SYSTEM TestFirstAgentFB (* System Configuration *)
  (* Standard: 61499-1 *)
  (* Version 0.3, 2003-12-05, JHC, Rockwell Automation, Renamed from NEWSYSTEM. *)
  (* Version 0.2, 2002-11-05, JHC, Rockwell Automation, Fixed missing (empty) FBD in Application. *)
  (* Version 0.1, 2002-01-17, JHC, Rockwell Automation, Minor cleanup *)
  (* Version 0.0, 2000-05-27, JHC, Rockwell Automation *)
  APPLICATION APP1
  END_APPLICATION
  DEVICE MyPLC : FRAME_DEVICE(BOUNDS := [1100,100,500,500], GRID := [1,1])
    RESOURCE MyProcessor : PANEL_RESOURCE(ROWS := 4, COLS := 4)
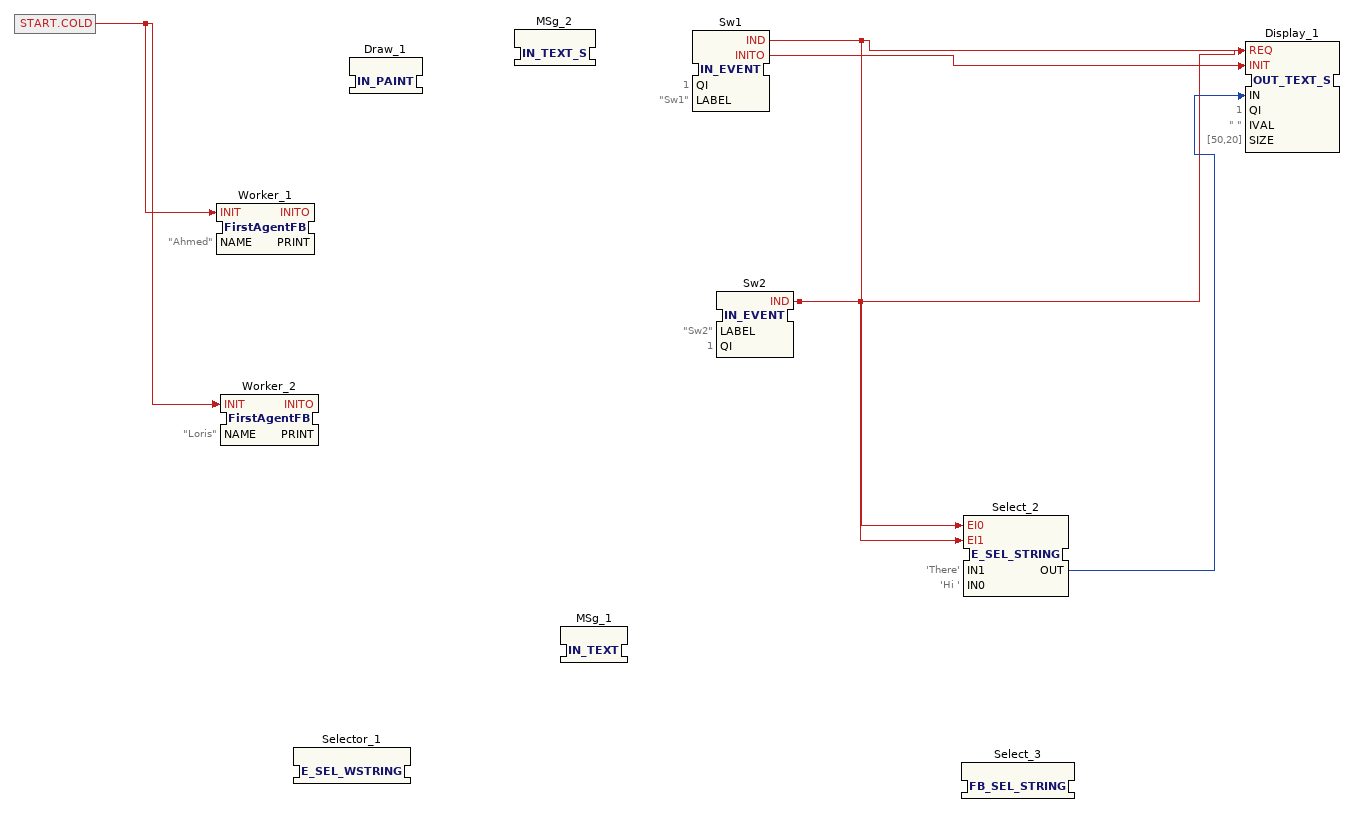
      FBS
        Worker_1 : FirstAgentFB(NAME := "Ahmed");
        Worker_2 : FirstAgentFB(NAME := "Loris");
        Display_1 : OUT_TEXT_S(QI := 1, IVAL := " ", SIZE := [50,20]);
        Sw1 : IN_EVENT(QI := 1, LABEL := "Sw1");
        MSg_1 : IN_TEXT;
        Draw_1 : IN_PAINT;
        Selector_1 : E_SEL_WSTRING;
        MSg_2 : IN_TEXT_S;
        Select_2 : E_SEL_STRING(IN1 := 'There', IN0 := 'Hi ');
        Sw2 : IN_EVENT(LABEL := "Sw2", QI := 1);
        Select_3 : FB_SEL_STRING;
      END_FBS
      EVENT_CONNECTIONS
        Sw1.IND TO Display_1.REQ;
        Sw1.INITO TO Display_1.INIT;
        Sw1.IND TO Select_2.EI0;
        Sw2.IND TO Select_2.EI1;
        Sw2.IND TO Display_1.REQ;
        START.COLD TO Worker_1.INIT;
        START.COLD TO Worker_2.INIT;
      END_CONNECTIONS
      DATA_CONNECTIONS
        Select_2.OUT TO Display_1.IN;
      END_CONNECTIONS
    END_RESOURCE
  END_DEVICE
END_SYSTEM
